TYPE ST_HMI_MapItem : 
STRUCT
	sName: WSTRING(127);
	sDescription: WSTRING(127);
	sPosition: WSTRING(127);
	nStatus: INT;
END_STRUCT
END_TYPE

(* stored: DUT ST_HMI_MapItem: Id 76f0fae0-218d-48c4-92a3-6a1581d7a270 *)
